RoboDK station: WORKING_EXAMPLE.rdk

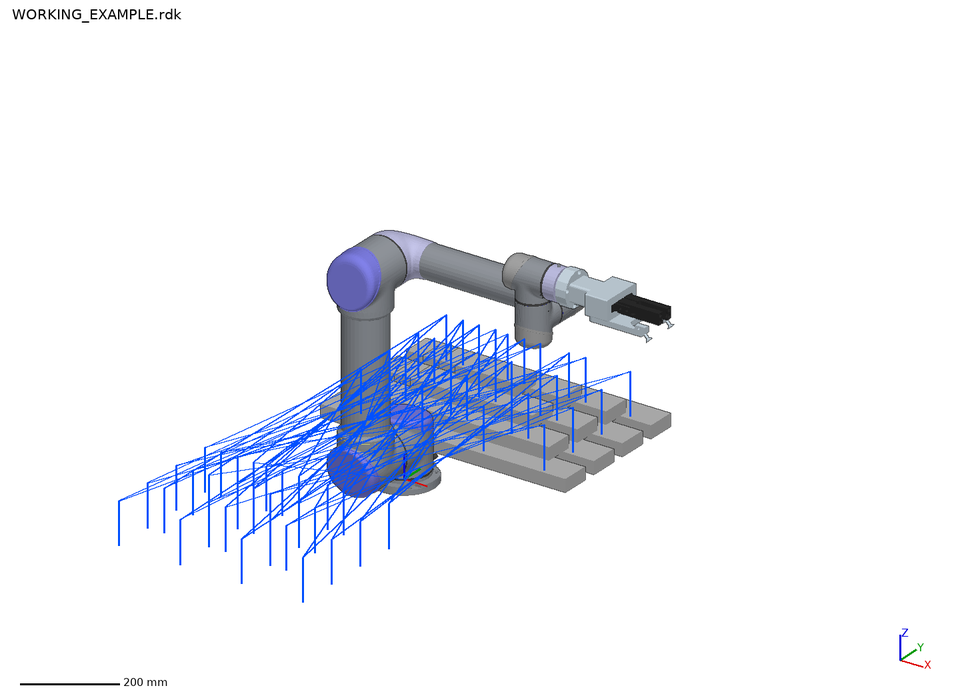
[picture v0: the station drawn from its stored meshes, robots at their saved joint values, targets as dots, program paths as lines]
Station WORKING_EXAMPLE (saved by RoboDK 5.2.1). Poses are relative to the parent item; angles as X-Y-Z fixed-axis rotations.
Station parameters (name, value as stored): Gripper, 0, CollisionFreePlanner, UR5, CollisionFreePlanner-Rob UR5
  - frame UR5 Base at (0, 0, 0) mm
    - robot UR5: 6 axes, payload 5 kg, reach 850 mm, repeatability 0.1 mm, weight 18.4 kg
        modified DH rows (alpha deg, a mm, theta deg, d mm): 0, 0, 0, 89.2; 90, 0, 180, 0; 0, 425, 0, 0; 0, 392.43, 0, 109; -90, 0, 0, 93.65; 90, 0, 180, 82
        joint limits [-360, -180, -180, -360, -360, -360] to [360, 0, 180, 0, 360, 360]; home [0, -90, -90, 0, 90, 0]; saved at [0, -90, -90, 0, 90, 0]
      - tool Gripper, TCP at (0, 0, 240) mm, rotated rx 0 ry 0 rz -90 deg, size 100 x 89.2 x 240.5 mm
    - frame FrameN at (0, 0, 0) mm
      - target csv_data-0 (Cartesian target) at (-26, 357, 183) mm, rotated rx 180 ry 0 rz 180 deg; joints [0, -90, -90, 0, 90, 0] of UR5
      - target csv_data-1 (Cartesian target) at (-26, 357, 83) mm, rotated rx 180 ry 0 rz 180 deg; joints [0, -90, -90, 0, 90, 0] of UR5
      - target csv_data-2 (Cartesian target) at (-26, 357, 183) mm, rotated rx 180 ry 0 rz 180 deg; joints [0, -90, -90, 0, 90, 0] of UR5
      - target csv_data-3 (Cartesian target) at (-301, -567, 93) mm, rotated rx 180 ry 0 rz 180 deg; joints [0, -90, -90, 0, 90, 0] of UR5
      - target csv_data-4 (Cartesian target) at (-301, -567, -7) mm, rotated rx 180 ry 0 rz 180 deg; joints [0, -90, -90, 0, 90, 0] of UR5
      - target csv_data-5 (Cartesian target) at (-301, -567, 93) mm, rotated rx 180 ry 0 rz 180 deg; joints [0, -90, -90, 0, 90, 0] of UR5
      - target csv_data-6 (Cartesian target) at (49, 407, 153) mm, rotated rx 180 ry 0 rz 0 deg; joints [0, -90, -90, 0, 90, 0] of UR5
      - target csv_data-7 (Cartesian target) at (49, 407, 53) mm, rotated rx 180 ry 0 rz 0 deg; joints [0, -90, -90, 0, 90, 0] of UR5
      - target csv_data-8 (Cartesian target) at (49, 407, 153) mm, rotated rx 180 ry 0 rz 0 deg; joints [0, -90, -90, 0, 90, 0] of UR5
      - target csv_data-9 (Cartesian target) at (-151, -567, 93) mm, rotated rx 180 ry 0 rz 180 deg; joints [0, -90, -90, 0, 90, 0] of UR5
      - target csv_data-10 (Cartesian target) at (-151, -567, -7) mm, rotated rx 180 ry 0 rz 180 deg; joints [0, -90, -90, 0, 90, 0] of UR5
      - target csv_data-11 (Cartesian target) at (-151, -567, 93) mm, rotated rx 180 ry 0 rz 180 deg; joints [0, -90, -90, 0, 90, 0] of UR5
      - target csv_data-12 (Cartesian target) at (-101, 407, 153) mm, rotated rx 180 ry 0 rz 180 deg; joints [0, -90, -90, 0, 90, 0] of UR5
      - target csv_data-13 (Cartesian target) at (-101, 407, 53) mm, rotated rx 180 ry 0 rz 180 deg; joints [0, -90, -90, 0, 90, 0] of UR5
      - target csv_data-14 (Cartesian target) at (-101, 407, 153) mm, rotated rx 180 ry 0 rz 180 deg; joints [0, -90, -90, 0, 90, 0] of UR5
      - target csv_data-15 (Cartesian target) at (-1, -567, 93) mm, rotated rx 180 ry 0 rz 180 deg; joints [0, -90, -90, 0, 90, 0] of UR5
      - target csv_data-16 (Cartesian target) at (-1, -567, -7) mm, rotated rx 180 ry 0 rz 180 deg; joints [0, -90, -90, 0, 90, 0] of UR5
      - target csv_data-17 (Cartesian target) at (-1, -567, 93) mm, rotated rx 180 ry 0 rz 180 deg; joints [0, -90, -90, 0, 90, 0] of UR5
      - target csv_data-18 (Cartesian target) at (49, 307, 153) mm, rotated rx 180 ry 0 rz 0 deg; joints [0, -90, -90, 0, 90, 0] of UR5
      - target csv_data-19 (Cartesian target) at (49, 307, 53) mm, rotated rx 180 ry 0 rz 0 deg; joints [0, -90, -90, 0, 90, 0] of UR5
      - target csv_data-20 (Cartesian target) at (49, 307, 153) mm, rotated rx 180 ry 0 rz 0 deg; joints [0, -90, -90, 0, 90, 0] of UR5
      - target csv_data-21 (Cartesian target) at (149, -567, 93) mm, rotated rx 180 ry 0 rz 0 deg; joints [0, -90, -90, 0, 90, 0] of UR5
      - target csv_data-22 (Cartesian target) at (149, -567, -7) mm, rotated rx 180 ry 0 rz 0 deg; joints [0, -90, -90, 0, 90, 0] of UR5
      - target csv_data-23 (Cartesian target) at (149, -567, 93) mm, rotated rx 180 ry 0 rz 0 deg; joints [0, -90, -90, 0, 90, 0] of UR5
      - target csv_data-24 (Cartesian target) at (-101, 307, 153) mm, rotated rx 180 ry 0 rz 180 deg; joints [0, -90, -90, 0, 90, 0] of UR5
      - target csv_data-25 (Cartesian target) at (-101, 307, 53) mm, rotated rx 180 ry 0 rz 180 deg; joints [0, -90, -90, 0, 90, 0] of UR5
      - target csv_data-26 (Cartesian target) at (-101, 307, 153) mm, rotated rx 180 ry 0 rz 180 deg; joints [0, -90, -90, 0, 90, 0] of UR5
      - target csv_data-27 (Cartesian target) at (-301, -467, 93) mm, rotated rx 180 ry 0 rz 180 deg; joints [0, -90, -90, 0, 90, 0] of UR5
      - target csv_data-28 (Cartesian target) at (-301, -467, -7) mm, rotated rx 180 ry 0 rz 180 deg; joints [0, -90, -90, 0, 90, 0] of UR5
      - target csv_data-29 (Cartesian target) at (-301, -467, 93) mm, rotated rx 180 ry 0 rz 180 deg; joints [0, -90, -90, 0, 90, 0] of UR5
      - target csv_data-30 (Cartesian target) at (124, 457, 123) mm, rotated rx 180 ry 0 rz 0 deg; joints [0, -90, -90, 0, 90, 0] of UR5
      - target csv_data-31 (Cartesian target) at (124, 457, 23) mm, rotated rx 180 ry 0 rz 0 deg; joints [0, -90, -90, 0, 90, 0] of UR5
      - target csv_data-32 (Cartesian target) at (124, 457, 123) mm, rotated rx 180 ry 0 rz 0 deg; joints [0, -90, -90, 0, 90, 0] of UR5
      - target csv_data-33 (Cartesian target) at (-151, -467, 93) mm, rotated rx 180 ry 0 rz 180 deg; joints [0, -90, -90, 0, 90, 0] of UR5
      - target csv_data-34 (Cartesian target) at (-151, -467, -7) mm, rotated rx 180 ry 0 rz 180 deg; joints [0, -90, -90, 0, 90, 0] of UR5
      - target csv_data-35 (Cartesian target) at (-151, -467, 93) mm, rotated rx 180 ry 0 rz 180 deg; joints [0, -90, -90, 0, 90, 0] of UR5
      - target csv_data-36 (Cartesian target) at (-26, 457, 123) mm, rotated rx 180 ry 0 rz 180 deg; joints [0, -90, -90, 0, 90, 0] of UR5
      - target csv_data-37 (Cartesian target) at (-26, 457, 23) mm, rotated rx 180 ry 0 rz 180 deg; joints [0, -90, -90, 0, 90, 0] of UR5
      - target csv_data-38 (Cartesian target) at (-26, 457, 123) mm, rotated rx 180 ry 0 rz 180 deg; joints [0, -90, -90, 0, 90, 0] of UR5
      - target csv_data-39 (Cartesian target) at (-1, -467, 93) mm, rotated rx 180 ry 0 rz 180 deg; joints [0, -90, -90, 0, 90, 0] of UR5
      - target csv_data-40 (Cartesian target) at (-1, -467, -7) mm, rotated rx 180 ry 0 rz 180 deg; joints [0, -90, -90, 0, 90, 0] of UR5
      - target csv_data-41 (Cartesian target) at (-1, -467, 93) mm, rotated rx 180 ry 0 rz 180 deg; joints [0, -90, -90, 0, 90, 0] of UR5
      - target csv_data-42 (Cartesian target) at (-176, 457, 123) mm, rotated rx 180 ry 0 rz 180 deg; joints [0, -90, -90, 0, 90, 0] of UR5
      - target csv_data-43 (Cartesian target) at (-176, 457, 23) mm, rotated rx 180 ry 0 rz 180 deg; joints [0, -90, -90, 0, 90, 0] of UR5
      - target csv_data-44 (Cartesian target) at (-176, 457, 123) mm, rotated rx 180 ry 0 rz 180 deg; joints [0, -90, -90, 0, 90, 0] of UR5
      - target csv_data-45 (Cartesian target) at (149, -467, 93) mm, rotated rx 180 ry 0 rz 0 deg; joints [0, -90, -90, 0, 90, 0] of UR5
      - target csv_data-46 (Cartesian target) at (149, -467, -7) mm, rotated rx 180 ry 0 rz 0 deg; joints [0, -90, -90, 0, 90, 0] of UR5
      - target csv_data-47 (Cartesian target) at (149, -467, 93) mm, rotated rx 180 ry 0 rz 0 deg; joints [0, -90, -90, 0, 90, 0] of UR5
      - target csv_data-48 (Cartesian target) at (124, 357, 123) mm, rotated rx 180 ry 0 rz 0 deg; joints [0, -90, -90, 0, 90, 0] of UR5
      - target csv_data-49 (Cartesian target) at (124, 357, 23) mm, rotated rx 180 ry 0 rz 0 deg; joints [0, -90, -90, 0, 90, 0] of UR5
      - target csv_data-50 (Cartesian target) at (124, 357, 123) mm, rotated rx 180 ry 0 rz 0 deg; joints [0, -90, -90, 0, 90, 0] of UR5
      - target csv_data-51 (Cartesian target) at (-301, -367, 93) mm, rotated rx 180 ry 0 rz 180 deg; joints [0, -90, -90, 0, 90, 0] of UR5
      - target csv_data-52 (Cartesian target) at (-301, -367, -7) mm, rotated rx 180 ry 0 rz 180 deg; joints [0, -90, -90, 0, 90, 0] of UR5
      - target csv_data-53 (Cartesian target) at (-301, -367, 93) mm, rotated rx 180 ry 0 rz 180 deg; joints [0, -90, -90, 0, 90, 0] of UR5
      - target csv_data-54 (Cartesian target) at (-26, 357, 123) mm, rotated rx 180 ry 0 rz 180 deg; joints [0, -90, -90, 0, 90, 0] of UR5
      - target csv_data-55 (Cartesian target) at (-26, 357, 23) mm, rotated rx 180 ry 0 rz 180 deg; joints [0, -90, -90, 0, 90, 0] of UR5
      - target csv_data-56 (Cartesian target) at (-26, 357, 123) mm, rotated rx 180 ry 0 rz 180 deg; joints [0, -90, -90, 0, 90, 0] of UR5
      - target csv_data-57 (Cartesian target) at (-151, -367, 93) mm, rotated rx 180 ry 0 rz 180 deg; joints [0, -90, -90, 0, 90, 0] of UR5
      - target csv_data-58 (Cartesian target) at (-151, -367, -7) mm, rotated rx 180 ry 0 rz 180 deg; joints [0, -90, -90, 0, 90, 0] of UR5
      - target csv_data-59 (Cartesian target) at (-151, -367, 93) mm, rotated rx 180 ry 0 rz 180 deg; joints [0, -90, -90, 0, 90, 0] of UR5
      - target csv_data-60 (Cartesian target) at (-176, 357, 123) mm, rotated rx 180 ry 0 rz 180 deg; joints [0, -90, -90, 0, 90, 0] of UR5
      - target csv_data-61 (Cartesian target) at (-176, 357, 23) mm, rotated rx 180 ry 0 rz 180 deg; joints [0, -90, -90, 0, 90, 0] of UR5
      - target csv_data-62 (Cartesian target) at (-176, 357, 123) mm, rotated rx 180 ry 0 rz 180 deg; joints [0, -90, -90, 0, 90, 0] of UR5
      - target csv_data-63 (Cartesian target) at (-1, -367, 93) mm, rotated rx 180 ry 0 rz 180 deg; joints [0, -90, -90, 0, 90, 0] of UR5
      - target csv_data-64 (Cartesian target) at (-1, -367, -7) mm, rotated rx 180 ry 0 rz 180 deg; joints [0, -90, -90, 0, 90, 0] of UR5
      - target csv_data-65 (Cartesian target) at (-1, -367, 93) mm, rotated rx 180 ry 0 rz 180 deg; joints [0, -90, -90, 0, 90, 0] of UR5
      - target csv_data-66 (Cartesian target) at (124, 257, 123) mm, rotated rx 180 ry 0 rz 0 deg; joints [0, -90, -90, 0, 90, 0] of UR5
      - target csv_data-67 (Cartesian target) at (124, 257, 23) mm, rotated rx 180 ry 0 rz 0 deg; joints [0, -90, -90, 0, 90, 0] of UR5
      - target csv_data-68 (Cartesian target) at (124, 257, 123) mm, rotated rx 180 ry 0 rz 0 deg; joints [0, -90, -90, 0, 90, 0] of UR5
      - target csv_data-69 (Cartesian target) at (149, -367, 93) mm, rotated rx 180 ry 0 rz 0 deg; joints [0, -90, -90, 0, 90, 0] of UR5
      - target csv_data-70 (Cartesian target) at (149, -367, -7) mm, rotated rx 180 ry 0 rz 0 deg; joints [0, -90, -90, 0, 90, 0] of UR5
      - target csv_data-71 (Cartesian target) at (149, -367, 93) mm, rotated rx 180 ry 0 rz 0 deg; joints [0, -90, -90, 0, 90, 0] of UR5
      - target csv_data-72 (Cartesian target) at (-26, 257, 123) mm, rotated rx 180 ry 0 rz 180 deg; joints [0, -90, -90, 0, 90, 0] of UR5
      - target csv_data-73 (Cartesian target) at (-26, 257, 23) mm, rotated rx 180 ry 0 rz 180 deg; joints [0, -90, -90, 0, 90, 0] of UR5
      - target csv_data-74 (Cartesian target) at (-26, 257, 123) mm, rotated rx 180 ry 0 rz 180 deg; joints [0, -90, -90, 0, 90, 0] of UR5
      - target csv_data-75 (Cartesian target) at (-301, -267, 93) mm, rotated rx 180 ry 0 rz 180 deg; joints [0, -90, -90, 0, 90, 0] of UR5
      - target csv_data-76 (Cartesian target) at (-301, -267, -7) mm, rotated rx 180 ry 0 rz 180 deg; joints [0, -90, -90, 0, 90, 0] of UR5
      - target csv_data-77 (Cartesian target) at (-301, -267, 93) mm, rotated rx 180 ry 0 rz 180 deg; joints [0, -90, -90, 0, 90, 0] of UR5
      - target csv_data-78 (Cartesian target) at (-176, 257, 123) mm, rotated rx 180 ry 0 rz 180 deg; joints [0, -90, -90, 0, 90, 0] of UR5
      - target csv_data-79 (Cartesian target) at (-176, 257, 23) mm, rotated rx 180 ry 0 rz 180 deg; joints [0, -90, -90, 0, 90, 0] of UR5
      - target csv_data-80 (Cartesian target) at (-176, 257, 123) mm, rotated rx 180 ry 0 rz 180 deg; joints [0, -90, -90, 0, 90, 0] of UR5
      - target csv_data-81 (Cartesian target) at (-151, -267, 93) mm, rotated rx 180 ry 0 rz 180 deg; joints [0, -90, -90, 0, 90, 0] of UR5
      - target csv_data-82 (Cartesian target) at (-151, -267, -7) mm, rotated rx 180 ry 0 rz 180 deg; joints [0, -90, -90, 0, 90, 0] of UR5
      - target csv_data-83 (Cartesian target) at (-151, -267, 93) mm, rotated rx 180 ry 0 rz 180 deg; joints [0, -90, -90, 0, 90, 0] of UR5
      - target csv_data-84 (Cartesian target) at (199, 507, 93) mm, rotated rx 180 ry 0 rz 0 deg; joints [0, -90, -90, 0, 90, 0] of UR5
      - target csv_data-85 (Cartesian target) at (199, 507, -7) mm, rotated rx 180 ry 0 rz 0 deg; joints [0, -90, -90, 0, 90, 0] of UR5
      - target csv_data-86 (Cartesian target) at (199, 507, 93) mm, rotated rx 180 ry 0 rz 0 deg; joints [0, -90, -90, 0, 90, 0] of UR5
      - target csv_data-87 (Cartesian target) at (-1, -267, 93) mm, rotated rx 180 ry 0 rz 180 deg; joints [0, -90, -90, 0, 90, 0] of UR5
      - target csv_data-88 (Cartesian target) at (-1, -267, -7) mm, rotated rx 180 ry 0 rz 180 deg; joints [0, -90, -90, 0, 90, 0] of UR5
      - target csv_data-89 (Cartesian target) at (-1, -267, 93) mm, rotated rx 180 ry 0 rz 180 deg; joints [0, -90, -90, 0, 90, 0] of UR5
      - target csv_data-90 (Cartesian target) at (49, 507, 93) mm, rotated rx 180 ry 0 rz 0 deg; joints [0, -90, -90, 0, 90, 0] of UR5
      - target csv_data-91 (Cartesian target) at (49, 507, -7) mm, rotated rx 180 ry 0 rz 0 deg; joints [0, -90, -90, 0, 90, 0] of UR5
      - target csv_data-92 (Cartesian target) at (49, 507, 93) mm, rotated rx 180 ry 0 rz 0 deg; joints [0, -90, -90, 0, 90, 0] of UR5
      - target csv_data-93 (Cartesian target) at (149, -267, 93) mm, rotated rx 180 ry 0 rz 0 deg; joints [0, -90, -90, 0, 90, 0] of UR5
      - target csv_data-94 (Cartesian target) at (149, -267, -7) mm, rotated rx 180 ry 0 rz 0 deg; joints [0, -90, -90, 0, 90, 0] of UR5
      - target csv_data-95 (Cartesian target) at (149, -267, 93) mm, rotated rx 180 ry 0 rz 0 deg; joints [0, -90, -90, 0, 90, 0] of UR5
      - target csv_data-96 (Cartesian target) at (-101, 507, 93) mm, rotated rx 180 ry 0 rz 180 deg; joints [0, -90, -90, 0, 90, 0] of UR5
      - target csv_data-97 (Cartesian target) at (-101, 507, -7) mm, rotated rx 180 ry 0 rz 180 deg; joints [0, -90, -90, 0, 90, 0] of UR5
      - target csv_data-98 (Cartesian target) at (-101, 507, 93) mm, rotated rx 180 ry 0 rz 180 deg; joints [0, -90, -90, 0, 90, 0] of UR5
      - target csv_data-99 (Cartesian target) at (-226, -517, 123) mm, rotated rx 180 ry 0 rz 180 deg; joints [0, -90, -90, 0, 90, 0] of UR5
      - target csv_data-100 (Cartesian target) at (-226, -517, 23) mm, rotated rx 180 ry 0 rz 180 deg; joints [0, -90, -90, 0, 90, 0] of UR5
      - target csv_data-101 (Cartesian target) at (-226, -517, 123) mm, rotated rx 180 ry 0 rz 180 deg; joints [0, -90, -90, 0, 90, 0] of UR5
      - target csv_data-102 (Cartesian target) at (-251, 507, 93) mm, rotated rx 180 ry 0 rz 180 deg; joints [0, -90, -90, 0, 90, 0] of UR5
      - target csv_data-103 (Cartesian target) at (-251, 507, -7) mm, rotated rx 180 ry 0 rz 180 deg; joints [0, -90, -90, 0, 90, 0] of UR5
      - target csv_data-104 (Cartesian target) at (-251, 507, 93) mm, rotated rx 180 ry 0 rz 180 deg; joints [0, -90, -90, 0, 90, 0] of UR5
      - target csv_data-105 (Cartesian target) at (-76, -517, 123) mm, rotated rx 180 ry 0 rz 180 deg; joints [0, -90, -90, 0, 90, 0] of UR5
      - target csv_data-106 (Cartesian target) at (-76, -517, 23) mm, rotated rx 180 ry 0 rz 180 deg; joints [0, -90, -90, 0, 90, 0] of UR5
      - target csv_data-107 (Cartesian target) at (-76, -517, 123) mm, rotated rx 180 ry 0 rz 180 deg; joints [0, -90, -90, 0, 90, 0] of UR5
      - target csv_data-108 (Cartesian target) at (199, 407, 93) mm, rotated rx 180 ry 0 rz 0 deg; joints [0, -90, -90, 0, 90, 0] of UR5
      - target csv_data-109 (Cartesian target) at (199, 407, -7) mm, rotated rx 180 ry 0 rz 0 deg; joints [0, -90, -90, 0, 90, 0] of UR5
      - target csv_data-110 (Cartesian target) at (199, 407, 93) mm, rotated rx 180 ry 0 rz 0 deg; joints [0, -90, -90, 0, 90, 0] of UR5
      - target csv_data-111 (Cartesian target) at (74, -517, 123) mm, rotated rx 180 ry 0 rz 0 deg; joints [0, -90, -90, 0, 90, 0] of UR5
      - target csv_data-112 (Cartesian target) at (74, -517, 23) mm, rotated rx 180 ry 0 rz 0 deg; joints [0, -90, -90, 0, 90, 0] of UR5
      - target csv_data-113 (Cartesian target) at (74, -517, 123) mm, rotated rx 180 ry 0 rz 0 deg; joints [0, -90, -90, 0, 90, 0] of UR5
      - target csv_data-114 (Cartesian target) at (49, 407, 93) mm, rotated rx 180 ry 0 rz 0 deg; joints [0, -90, -90, 0, 90, 0] of UR5
      - target csv_data-115 (Cartesian target) at (49, 407, -7) mm, rotated rx 180 ry 0 rz 0 deg; joints [0, -90, -90, 0, 90, 0] of UR5
      - target csv_data-116 (Cartesian target) at (49, 407, 93) mm, rotated rx 180 ry 0 rz 0 deg; joints [0, -90, -90, 0, 90, 0] of UR5
      - target csv_data-117 (Cartesian target) at (-226, -417, 123) mm, rotated rx 180 ry 0 rz 180 deg; joints [0, -90, -90, 0, 90, 0] of UR5
      - target csv_data-118 (Cartesian target) at (-226, -417, 23) mm, rotated rx 180 ry 0 rz 180 deg; joints [0, -90, -90, 0, 90, 0] of UR5
      - target csv_data-119 (Cartesian target) at (-226, -417, 123) mm, rotated rx 180 ry 0 rz 180 deg; joints [0, -90, -90, 0, 90, 0] of UR5
      - target csv_data-120 (Cartesian target) at (-101, 407, 93) mm, rotated rx 180 ry 0 rz 180 deg; joints [0, -90, -90, 0, 90, 0] of UR5
      - target csv_data-121 (Cartesian target) at (-101, 407, -7) mm, rotated rx 180 ry 0 rz 180 deg; joints [0, -90, -90, 0, 90, 0] of UR5
      - target csv_data-122 (Cartesian target) at (-101, 407, 93) mm, rotated rx 180 ry 0 rz 180 deg; joints [0, -90, -90, 0, 90, 0] of UR5
      - target csv_data-123 (Cartesian target) at (-76, -417, 123) mm, rotated rx 180 ry 0 rz 180 deg; joints [0, -90, -90, 0, 90, 0] of UR5
      - target csv_data-124 (Cartesian target) at (-76, -417, 23) mm, rotated rx 180 ry 0 rz 180 deg; joints [0, -90, -90, 0, 90, 0] of UR5
      - target csv_data-125 (Cartesian target) at (-76, -417, 123) mm, rotated rx 180 ry 0 rz 180 deg; joints [0, -90, -90, 0, 90, 0] of UR5
      - target csv_data-126 (Cartesian target) at (-251, 407, 93) mm, rotated rx 180 ry 0 rz 180 deg; joints [0, -90, -90, 0, 90, 0] of UR5
      - target csv_data-127 (Cartesian target) at (-251, 407, -7) mm, rotated rx 180 ry 0 rz 180 deg; joints [0, -90, -90, 0, 90, 0] of UR5
      - target csv_data-128 (Cartesian target) at (-251, 407, 93) mm, rotated rx 180 ry 0 rz 180 deg; joints [0, -90, -90, 0, 90, 0] of UR5
      - target csv_data-129 (Cartesian target) at (74, -417, 123) mm, rotated rx 180 ry 0 rz 0 deg; joints [0, -90, -90, 0, 90, 0] of UR5
      - target csv_data-130 (Cartesian target) at (74, -417, 23) mm, rotated rx 180 ry 0 rz 0 deg; joints [0, -90, -90, 0, 90, 0] of UR5
      - target csv_data-131 (Cartesian target) at (74, -417, 123) mm, rotated rx 180 ry 0 rz 0 deg; joints [0, -90, -90, 0, 90, 0] of UR5
      - target csv_data-132 (Cartesian target) at (199, 307, 93) mm, rotated rx 180 ry 0 rz 0 deg; joints [0, -90, -90, 0, 90, 0] of UR5
      - target csv_data-133 (Cartesian target) at (199, 307, -7) mm, rotated rx 180 ry 0 rz 0 deg; joints [0, -90, -90, 0, 90, 0] of UR5
      - target csv_data-134 (Cartesian target) at (199, 307, 93) mm, rotated rx 180 ry 0 rz 0 deg; joints [0, -90, -90, 0, 90, 0] of UR5
      - target csv_data-135 (Cartesian target) at (-226, -317, 123) mm, rotated rx 180 ry 0 rz 180 deg; joints [0, -90, -90, 0, 90, 0] of UR5
      - target csv_data-136 (Cartesian target) at (-226, -317, 23) mm, rotated rx 180 ry 0 rz 180 deg; joints [0, -90, -90, 0, 90, 0] of UR5
      - target csv_data-137 (Cartesian target) at (-226, -317, 123) mm, rotated rx 180 ry 0 rz 180 deg; joints [0, -90, -90, 0, 90, 0] of UR5
      - target csv_data-138 (Cartesian target) at (49, 307, 93) mm, rotated rx 180 ry 0 rz 0 deg; joints [0, -90, -90, 0, 90, 0] of UR5
      - target csv_data-139 (Cartesian target) at (49, 307, -7) mm, rotated rx 180 ry 0 rz 0 deg; joints [0, -90, -90, 0, 90, 0] of UR5
      - target csv_data-140 (Cartesian target) at (49, 307, 93) mm, rotated rx 180 ry 0 rz 0 deg; joints [0, -90, -90, 0, 90, 0] of UR5
      - target csv_data-141 (Cartesian target) at (-76, -317, 123) mm, rotated rx 180 ry 0 rz 180 deg; joints [0, -90, -90, 0, 90, 0] of UR5
      - target csv_data-142 (Cartesian target) at (-76, -317, 23) mm, rotated rx 180 ry 0 rz 180 deg; joints [0, -90, -90, 0, 90, 0] of UR5
      - target csv_data-143 (Cartesian target) at (-76, -317, 123) mm, rotated rx 180 ry 0 rz 180 deg; joints [0, -90, -90, 0, 90, 0] of UR5
      - target csv_data-144 (Cartesian target) at (-101, 307, 93) mm, rotated rx 180 ry 0 rz 180 deg; joints [0, -90, -90, 0, 90, 0] of UR5
      - target csv_data-145 (Cartesian target) at (-101, 307, -7) mm, rotated rx 180 ry 0 rz 180 deg; joints [0, -90, -90, 0, 90, 0] of UR5
      - target csv_data-146 (Cartesian target) at (-101, 307, 93) mm, rotated rx 180 ry 0 rz 180 deg; joints [0, -90, -90, 0, 90, 0] of UR5
      - target csv_data-147 (Cartesian target) at (74, -317, 123) mm, rotated rx 180 ry 0 rz 0 deg; joints [0, -90, -90, 0, 90, 0] of UR5
      - target csv_data-148 (Cartesian target) at (74, -317, 23) mm, rotated rx 180 ry 0 rz 0 deg; joints [0, -90, -90, 0, 90, 0] of UR5
      - target csv_data-149 (Cartesian target) at (74, -317, 123) mm, rotated rx 180 ry 0 rz 0 deg; joints [0, -90, -90, 0, 90, 0] of UR5
      - target csv_data-150 (Cartesian target) at (-251, 307, 93) mm, rotated rx 180 ry 0 rz 180 deg; joints [0, -90, -90, 0, 90, 0] of UR5
      - target csv_data-151 (Cartesian target) at (-251, 307, -7) mm, rotated rx 180 ry 0 rz 180 deg; joints [0, -90, -90, 0, 90, 0] of UR5
      - target csv_data-152 (Cartesian target) at (-251, 307, 93) mm, rotated rx 180 ry 0 rz 180 deg; joints [0, -90, -90, 0, 90, 0] of UR5
      - target csv_data-153 (Cartesian target) at (-151, -467, 153) mm, rotated rx 180 ry 0 rz 180 deg; joints [0, -90, -90, 0, 90, 0] of UR5
      - target csv_data-154 (Cartesian target) at (-151, -467, 53) mm, rotated rx 180 ry 0 rz 180 deg; joints [0, -90, -90, 0, 90, 0] of UR5
      - target csv_data-155 (Cartesian target) at (-151, -467, 153) mm, rotated rx 180 ry 0 rz 180 deg; joints [0, -90, -90, 0, 90, 0] of UR5
      - target csv_data-156 (Cartesian target) at (199, 207, 93) mm, rotated rx 180 ry 0 rz 0 deg; joints [0, -90, -90, 0, 90, 0] of UR5
      - target csv_data-157 (Cartesian target) at (199, 207, -7) mm, rotated rx 180 ry 0 rz 0 deg; joints [0, -90, -90, 0, 90, 0] of UR5
      - target csv_data-158 (Cartesian target) at (199, 207, 93) mm, rotated rx 180 ry 0 rz 0 deg; joints [0, -90, -90, 0, 90, 0] of UR5
      - target csv_data-159 (Cartesian target) at (-1, -467, 153) mm, rotated rx 180 ry 0 rz 180 deg; joints [0, -90, -90, 0, 90, 0] of UR5
      - target csv_data-160 (Cartesian target) at (-1, -467, 53) mm, rotated rx 180 ry 0 rz 180 deg; joints [0, -90, -90, 0, 90, 0] of UR5
      - target csv_data-161 (Cartesian target) at (-1, -467, 153) mm, rotated rx 180 ry 0 rz 180 deg; joints [0, -90, -90, 0, 90, 0] of UR5
      - target csv_data-162 (Cartesian target) at (49, 207, 93) mm, rotated rx 180 ry 0 rz 0 deg; joints [0, -90, -90, 0, 90, 0] of UR5
      - target csv_data-163 (Cartesian target) at (49, 207, -7) mm, rotated rx 180 ry 0 rz 0 deg; joints [0, -90, -90, 0, 90, 0] of UR5
      - target csv_data-164 (Cartesian target) at (49, 207, 93) mm, rotated rx 180 ry 0 rz 0 deg; joints [0, -90, -90, 0, 90, 0] of UR5
      - target csv_data-165 (Cartesian target) at (-151, -367, 153) mm, rotated rx 180 ry 0 rz 180 deg; joints [0, -90, -90, 0, 90, 0] of UR5
      - target csv_data-166 (Cartesian target) at (-151, -367, 53) mm, rotated rx 180 ry 0 rz 180 deg; joints [0, -90, -90, 0, 90, 0] of UR5
      - target csv_data-167 (Cartesian target) at (-151, -367, 153) mm, rotated rx 180 ry 0 rz 180 deg; joints [0, -90, -90, 0, 90, 0] of UR5
      - target csv_data-168 (Cartesian target) at (-101, 207, 93) mm, rotated rx 180 ry 0 rz 180 deg; joints [0, -90, -90, 0, 90, 0] of UR5
      - target csv_data-169 (Cartesian target) at (-101, 207, -7) mm, rotated rx 180 ry 0 rz 180 deg; joints [0, -90, -90, 0, 90, 0] of UR5
      - target csv_data-170 (Cartesian target) at (-101, 207, 93) mm, rotated rx 180 ry 0 rz 180 deg; joints [0, -90, -90, 0, 90, 0] of UR5
      - target csv_data-171 (Cartesian target) at (-1, -367, 153) mm, rotated rx 180 ry 0 rz 180 deg; joints [0, -90, -90, 0, 90, 0] of UR5
      - target csv_data-172 (Cartesian target) at (-1, -367, 53) mm, rotated rx 180 ry 0 rz 180 deg; joints [0, -90, -90, 0, 90, 0] of UR5
      - target csv_data-173 (Cartesian target) at (-1, -367, 153) mm, rotated rx 180 ry 0 rz 180 deg; joints [0, -90, -90, 0, 90, 0] of UR5
      - target csv_data-174 (Cartesian target) at (-251, 207, 93) mm, rotated rx 180 ry 0 rz 180 deg; joints [0, -90, -90, 0, 90, 0] of UR5
      - target csv_data-175 (Cartesian target) at (-251, 207, -7) mm, rotated rx 180 ry 0 rz 180 deg; joints [0, -90, -90, 0, 90, 0] of UR5
      - target csv_data-176 (Cartesian target) at (-251, 207, 93) mm, rotated rx 180 ry 0 rz 180 deg; joints [0, -90, -90, 0, 90, 0] of UR5
      - target csv_data-177 (Cartesian target) at (-76, -417, 183) mm, rotated rx 180 ry 0 rz 180 deg; joints [0, -90, -90, 0, 90, 0] of UR5
      - target csv_data-178 (Cartesian target) at (-76, -417, 83) mm, rotated rx 180 ry 0 rz 180 deg; joints [0, -90, -90, 0, 90, 0] of UR5
      - target csv_data-179 (Cartesian target) at (-76, -417, 183) mm, rotated rx 180 ry 0 rz 180 deg; joints [0, -90, -90, 0, 90, 0] of UR5
    - object Table at (-250, 600, 0) mm, rotated rx 0 ry 0 rz -180 deg, size 600 x 1350 x 100 mm, geometry from RhinoPart.ply
    - object Closed Brep_0 at (0, 0, 0) mm, size 150 x 70 x 30 mm
    - object Closed Brep_1 at (0, 0, 0) mm, size 150 x 70 x 30 mm
    - object Closed Brep_2 at (0, 0, 0) mm, size 150 x 70 x 30 mm
    - object Closed Brep_3 at (0, 0, 0) mm, size 150 x 70 x 30 mm
    - object Closed Brep_4 at (0, 0, 0) mm, size 150 x 70 x 30 mm
    - object Closed Brep_5 at (0, 0, 0) mm, size 150 x 70 x 30 mm
    - object Closed Brep_6 at (0, 0, 0) mm, size 150 x 70 x 30 mm
    - object Closed Brep_7 at (0, 0, 0) mm, size 150 x 70 x 30 mm
    - object Closed Brep_8 at (0, 0, 0) mm, size 150 x 70 x 30 mm
    - object Closed Brep_9 at (0, 0, 0) mm, size 150 x 70 x 30 mm
    - object Closed Brep_10 at (0, 0, 0) mm, size 150 x 70 x 30 mm
    - object Closed Brep_11 at (0, 0, 0) mm, size 150 x 70 x 30 mm
    - object Closed Brep_12 at (0, 0, 0) mm, size 150 x 70 x 30 mm
    - object Closed Brep_13 at (0, 0, 0) mm, size 150 x 70 x 30 mm
    - object Closed Brep_14 at (0, 0, 0) mm, size 150 x 70 x 30 mm
    - object Closed Brep_15 at (0, 0, 0) mm, size 150 x 70 x 30 mm
    - object Closed Brep_16 at (0, 0, 0) mm, size 150 x 70 x 30 mm
    - object Closed Brep_17 at (0, 0, 0) mm, size 150 x 70 x 30 mm
    - object Closed Brep_18 at (0, 0, 0) mm, size 150 x 70 x 30 mm
    - object Closed Brep_19 at (0, 0, 0) mm, size 150 x 70 x 30 mm
    - object Closed Brep_20 at (0, 0, 0) mm, size 150 x 70 x 30 mm
    - object Closed Brep_21 at (0, 0, 0) mm, size 150 x 70 x 30 mm
    - object Closed Brep_22 at (0, 0, 0) mm, size 150 x 70 x 30 mm
    - object Closed Brep_23 at (0, 0, 0) mm, size 150 x 70 x 30 mm
    - object Closed Brep_24 at (0, 0, 0) mm, size 150 x 70 x 30 mm
    - object Closed Brep_25 at (0, 0, 0) mm, size 150 x 70 x 30 mm
    - object Closed Brep_26 at (0, 0, 0) mm, size 150 x 70 x 30 mm
    - object Closed Brep_27 at (0, 0, 0) mm, size 150 x 70 x 30 mm
    - object Closed Brep_28 at (0, 0, 0) mm, size 150 x 70 x 30 mm
    - object Closed Brep_29 at (0, 0, 0) mm, size 150 x 70 x 30 mm
  - Python program Generate_csv_program (listed below)
  - Python program Import_Rhino_geometry (listed below)
  - program Main_Program (365 instructions, listed below)
  - program Attach (3 instructions, listed below)
  - program Detach (3 instructions, listed below)
  - program Return_Bricks (1 instructions, listed below)
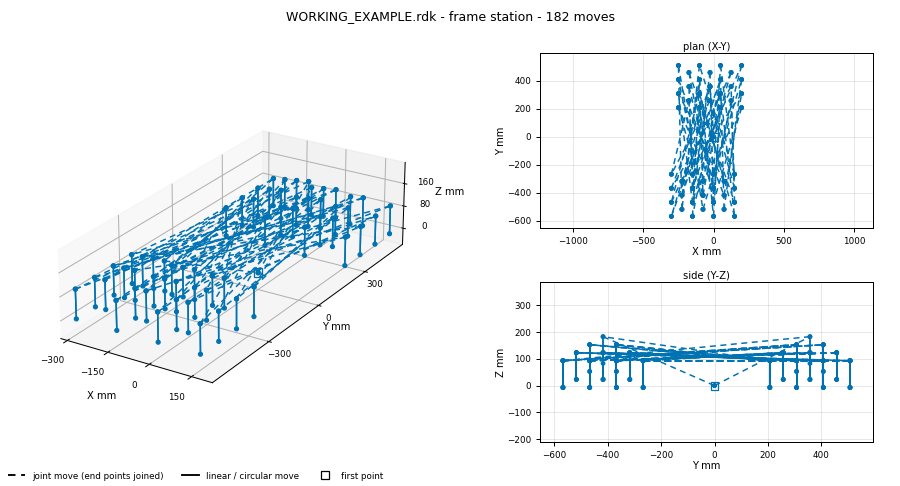
[picture p0: tool path of WORKING_EXAMPLE.rdk in frame station, 182 of 182 moves have a stored position in this frame; points joined in program order, loops and branches not executed]

--- Python program Generate_csv_program ---
# This macro can load CSV files in RoboDK. It also allows the user
# Supported types of files are:
#  1-Tool data : Tool.csv
#  2-Work object data: Work.csv
#  3-Target data: P_Var.csv
# This macro can also filter a given targets file

# Type help("robolink") or help("robodk") for more information
# Press F5 to run the script
# Visit: http://www.robodk.com/doc/PythonAPI/
# For RoboDK API documentation

# This script has been further developed by Job de Vogel
# It is based on the example ImportCSV_XYZWPR.py script

from robolink import *    # API to communicate with RoboDK
from robodk import *      # basic matrix operations

# Start communication with RoboDK
RDK = Robolink()

# Ask the user to select the robot (ignores the popup if only
ROBOT = RDK.ItemUserPick('Select a robot', ITEM_TYPE_ROBOT)

# Check if the user selected a robot
if not ROBOT.Valid():
    quit()

# Automatically retrieve active reference and tool
FRAME = ROBOT.getLink(ITEM_TYPE_FRAME)
TOOL = ROBOT.getLink(ITEM_TYPE_TOOL)

#FRAME = RDK.ItemUserPick('Select a reference frame', ITEM_TYPE_FRAME)
#TOOL = RDK.ItemUserPick('Select a tool', ITEM_TYPE_TOOL)

if not FRAME.Valid() or not TOOL.Valid():
    raise Exception("Select appropriate FRAME and TOOL references")

# Function to convert XYZWPR to a pose
# Important! Specify the order of rotation
def xyzwpr_to_pose(xyzwpr):
    x,y,z,rx,ry,rz = xyzwpr
    return transl(x,y,z)*rotz(rz*pi/180)*roty(ry*pi/180)*rotx(rx*pi/180)
    #return transl(x,y,z)*rotx(rx*pi/180)*roty(ry*pi/180)*rotz(rz*pi/180)
    #return KUKA_2_Pose(xyzwpr)

# Load P_Var.CSV data as a list of poses, including links to reference and tool frames
def load_targets(strfile):
    csvdata = LoadList(strfile, ',', codec)

    idxs = [] # row index of the csv data
    poses = [] # pose of the csv data, based on x,y,z,rx,ry,rz
    movetypes = [] # type of movement: linear (l) or joint (j)
    speeds = [] # joint speed of the robot
    subprogram_names = []

    """ EXTRACT EXTRA DATA
    HERE YOU INITIALIZE EXTRA VARIABLES THAT THE CSV DATA CONTAINS
    """

    # Iterate over the rows with instructions in the csv
    for i in range(0, len(csvdata)):
        # Extract the index of the instruction
        idxs.append(i)

        # Extract the pose data from the csv
        try:
            x,y,z,rx,ry,rz = csvdata[i][0:6]
            poses.append(xyzwpr_to_pose([x,y,z,rx,ry,rz]))
        except:
            print("No pose available to extract")
            return

        # Extract the speed data from the csv
        try:
            speed = csvdata[i][6]
            speeds.append(speed)
        except:
            speeds.append("")

        # Extract the movetypes from the csv
        try:
            movetype = csvdata[i][7]
            movetypes.append(movetype)
        except IndexError:
            movetypes.append("")

        # Extract the subprograms from the csv
        try:
            subprogram = csvdata[i][8]
            subprogram_names.append(subprogram)
        except:
            subprogram_names.append("")

        """ADD DATA
        HERE YOU EXTRACT OTHER DATA FROM THE CSV
        MAKE SURE YOU RETURN THE DATA AT THE END OF THIS DEFINITION

        ALWAYS ADD A TRY-EXCEPT STATEMENT IN CASE NO DATA IS
        AVAILABLE IN THE CSV
        """

    return idxs, poses, movetypes, speeds, subprogram_names

# Load the data from the CSV and add the instruction to the main program
def load_program_csv(strfile, program_name):
    # Get the data from .csv
    idxs, poses, movetypes, speeds, subprogram_names = load_targets(strfile)

    # Set the name for the csv
    csv_name = getFileName(strfile)
    csv_name = csv_name.replace('-','_').replace(' ','_')

    # Create a RDK program item
    program = RDK.Item(program_name, ITEM_TYPE_PROGRAM)

    # If the program already exists, delete it
    if program.Valid():
        program.Delete()

    # Add the main program to the robot
    program = RDK.AddProgram(program_name, ROBOT)

    # Set the frame and the tool to the main program
    program.setFrame(FRAME)
    program.setTool(TOOL)

    # Move the robot home
    ROBOT.MoveJ(ROBOT.JointsHome())
    program.MoveJ(ROBOT.JointsHome())

    # For each point from the csv, add the following instuction to the main program
    for idx, pose, movetype, speed, subprogram_name in zip(idxs, poses, movetypes, speeds, subprogram_names):

        #status = program.Update(1)
        #print(status)

        # Set the name of the point
        name = '%s-%i' % (csv_name, idx)

        # Create a target for the name
        target = RDK.Item(name, ITEM_TYPE_TARGET)

        # If the target already exists, delete it
        if target.Valid():
            target.Delete()

        # Add the target to the main program
        target = RDK.AddTarget(name, FRAME, ROBOT)
        target.setPose(pose)

        """ ADD INSTRUCTIONS
        FROM HERE ON, THE ROBOT WILL ADD THE INSTRUCTION FROM THE CSV TO THE PROGRAM
        CURRENTLY, THE INSTRUCTIONS ARE ADDED ACCORDING THE ORDER OF THE CSV COLUMNS
        """

        # Add the movement to the program
        # Overwrite to joint to avoid singularities:
        if movetype == "linear":
            try:
                program.MoveL(target)
            except:
                print('Warning: {} can not be reached. It will not be added to the program'.format(name))
        else:
            try:
                program.MoveJ(target)
            except:
                print('Warning: {} can not be reached. It will not be added to the program'.format(name))

        # Set a speed for the robot
        if speed:
            program.setSpeed(speed, speed)

        # Check if this csv row has a subprogram to run
        if subprogram_name:
            subprogram = RDK.Item(subprogram_name, ITEM_TYPE_PROGRAM)

            # If the subprogram does not yet exist, add it to the Robot tree
            if not subprogram.Valid():
                subprogram = RDK.AddProgram(subprogram_name, ROBOT)
                print("{} added to Robot".format(subprogram_name))

            program.RunInstruction(subprogram_name)

        """TO ADD INSTRUCTIONS:
        FROM HERE ON, YOU CAN ADD YOUR OWN INSTRUCTIONS TO THE ROBOT
        MAKE SURE YOU ADD THEM IN THE CORRECT ORDER

        TAKE A LOOK AT https://robodk.com/doc/en/PythonAPI/robolink.html TO SEE WHAT IS POSSIBLE
        """

    # Move the robot home
    program.MoveJ(ROBOT.JointsHome())
    print("{} has been updated!".format(program_name))

# Run the robot simulation
# The run_simulation function does the same as load_program_csv but it doesn't load the program
# to RoboDK. If you only want the Robot to do something, use ROBOT.function() instead of program.function()
# If the program already exists in the tree, it will directly use those instructions,
# to make use of collision detection
def run_simulation(strfile, program_name):
    # Load the data from the csv file
    idxs, poses, movetypes, speeds, subprogram_names = load_targets(strfile)

    # Set the frame and tool of the robot
    ROBOT.setFrame(FRAME)
    ROBOT.setTool(TOOL)

    # Return to home
    ROBOT.MoveJ(ROBOT.JointsHome())

    # Check if program is already added to the robot tree
    # If that is the case, run the instructions directly from the tree
    # Else, robot may execute script without proper collision avoidance
    program = RDK.Item(program_name, ITEM_TYPE_PROGRAM)
    if program.Valid():
        program.RunCode()
        return

    for idx, pose, movetype, speed, subprogram_name in zip(idxs, poses, movetypes, speeds, subprogram_names):
        # Move the robot according to movetype, if no movetype available, do a joint move
        # Overwrite to joint to avoid singularities:
        if movetype == "linear":
            try:
                ROBOT.MoveL(pose)
            except TargetReachError:
                RDK.ShowMessage('Target %i can not be reached' % idx, False)
        else:
            try:
                ROBOT.MoveJ(pose)
            except TargetReachError:
                RDK.ShowMessage('Target %i can not be reached' % idx, False)

        """
        IF YOU ADD INSTRUCTIONS TO THE LOAD_PROGRAM_CSV FUNCTION,
        YOU WILL ALSO NEED TO ADD THEM TO THE RUN_SIMULATION FUNCTION.
        """

        # If there is a speed available, set the linear and joint speed
        if speed:
            print("Set speed to {} m/s".format(speed))
            ROBOT.setSpeed(speed, speed)

        # If a subprogram should be run, run the subprogram
        if subprogram_name:
            subprogram = RDK.Item(subprogram_name, ITEM_TYPE_PROGRAM)

            if subprogram.Valid():
                print("Robot is running {}".format(subprogram_name))
                subprogram.RunCode()
            else:
                print("{} is not valid, the subprogram will be skipped".format(subprogram_name))

    # Return to home
    ROBOT.MoveJ(ROBOT.JointsHome())

######################################### -- MAIN -- ################################################
# Force just moving the robot after double clicking:
#load_targets_move(CSV_FILE)
#quit()

# Specify file codec
codec = 'utf-8' #'ISO-8859-1'

# SPECIFY YOU CSV FILE HERE:
CSV_FILE = r"" # Make sure you add r in front of your string to get a raw string as filepath
SELECT_CSV = mbox('Please select your csv file, you can also specify your csv directory in the generate_csv_program script (line 266)', 'Select')

if SELECT_CSV and not CSV_FILE:
    # No CSV has been specified in line 266, select manually
    CSV_FILE = getOpenFile(RDK.getParam('PATH_OPENSTATION'))
elif not SELECT_CSV and not CSV_FILE:
    # User wants to cancel
    quit()

# PROGRAM/SIMULATION SETTINGS:
MAKE_GUI_PROGRAM = False
SIMULATION_SPEED = 1
PROGRAM_NAME = "Main_Program"

ROBOT.setFrame(FRAME)
ROBOT.setTool(TOOL)

RDK.setSimulationSpeed(SIMULATION_SPEED)

if RDK.RunMode() == RUNMODE_SIMULATE:
    MAKE_GUI_PROGRAM = True
    if CSV_FILE:
        MAKE_GUI_PROGRAM = mbox('Do you want to create a new program? If not, the robot will execute a simulation. If the program does not exist in the RoboDK, collisions may occur!', 'Yes', 'No')
else:
    # If we run in program generation mode just move the robot
    MAKE_GUI_PROGRAM = False

if MAKE_GUI_PROGRAM:
    RDK.Render(False) # Faster if we turn render off
    load_program_csv(CSV_FILE, PROGRAM_NAME) # HERE THE CSV DATA IS LOADED!!!
else:
    run_simulation(CSV_FILE, PROGRAM_NAME) # HERE WE START RUNNING THE PROJECT!!!

--- Python program Import_Rhino_geometry ---
# Type help("robolink") or help("robodk") for more information
# Press F5 to run the script
# Documentation: https://robodk.com/doc/en/RoboDK-API.html
# Reference:     https://robodk.com/doc/en/PythonAPI/index.html

# This script has been developed by Job de Vogel
from robolink import *    # RoboDK API
from robodk import *      # Robot toolbox

RDK = Robolink()

# Ask the user to select the robot (ignores the popup if only
ROBOT = RDK.ItemUserPick('Select a robot', ITEM_TYPE_ROBOT)

# Check if the user selected a robot
if not ROBOT.Valid():
    quit()

# Read the csv with geometry
# First column in csv indicates type (v: vertex, o: order, n: name)
def load_csv_data(strfile):
    csv_file = LoadList(strfile, ',', codec)

    # Store the vertex data, vertex order and name in dict
    vertex_data = {}
    vertex_order = {}
    names = {}

    # For every csv line, check the data type and store value accordingly
    i = 0
    for line in csv_file:
        # Check if geom key in dict contains list, if not create it
        try:
            data = vertex_data[i]
            data = vertex_order[i]
        except KeyError:
            vertex_data[i] = []
            vertex_order[i] = []

        datatype = line[0]
        if datatype == 'v':
            vertex_data[i].append(line[1:])
        elif datatype == 'o':
            vertex_order[i].append(line[1:])
        elif datatype == 'n':
            names[i] = line[1]
            i +=1

    return vertex_data, vertex_order, names

# Create a list that contains all the vertices according to the vertexorder of the shape
def structure_vertexData(vertex_data: list, vertex_order: list):
    data = []
    for order in vertex_order:
        for vertex in order:
            data.append(vertex_data[int(vertex)])

    return data

# Create an RDK item that contains the shape
# The function will copy the shape to clipboard, it can be later pasted to frame using frame.Paste()
def create_shape(name, vertices):
    obj = RDK.Item(name, ITEM_TYPE_OBJECT)

    # If obj already exist, delete previous version
    if obj.Valid():
        obj.Delete()

    # Create a new shape for the obj
    obj = obj.AddShape(vertices)
    obj.setName(name)

    # Copy to paste after return
    obj.Copy()
    obj.Delete()
    return

######################################### -- MAIN -- ################################################
# Specify file codec
codec = 'utf-8' #'ISO-8859-1'

# SPECIFY YOU CSV FILE HERE:
objects_csv_file = r"" # Make sure you add r in front of your string to get a raw string for your filepath
SELECT_CSV = mbox('Please select your csv file that contains your geometry data and frame data. (You can also specify a path in the script in line 83)', 'Select')

if SELECT_CSV and not objects_csv_file:
    # No CSV has been specified in line 83, select manually
    objects_csv_file = getOpenFile(RDK.getParam('PATH_OPENSTATION'))

    if not objects_csv_file:
        quit()
elif not SELECT_CSV and not objects_csv_file:
    # User does not wants to cancel
    quit()

# HERE YOU CAN DEFINE WHERE THE OBJECTS SHOULD BE PASTED:
frame_name = 'UR5 Base' # Name of the frame where your geometry should be added
ROBOT_frame = RDK.Item(frame_name, ITEM_TYPE_FRAME)

if ROBOT_frame.Valid():
    mbox('Your geometry will be added to {}. You can change the frame in script line 97.'.format(frame_name), 'Okay')
else:
    ROBOT.getLink(ITEM_TYPE_FRAME)
    mbox('Your selected frame does not exist in the tree. Frame will be changed to standard Robot frame. Please change in script line 97.', 'Okay')

# Load the geometry csv
geometries = load_csv_data(objects_csv_file)

vertex_data = geometries[0].values()
vertex_order = geometries[1].values()
geom_names = geometries[2].values()

for i, (vertices, indices, geom_name) in enumerate(zip(vertex_data, vertex_order, geom_names)):
    geom_vertices = structure_vertexData(vertices, indices)

    #name = "Geom_{}".format(i)
    create_shape(geom_name, geom_vertices)

    ROBOT_frame.Paste()
    print("{} added to Robot tree".format(geom_name))

--- program Main_Program (robot UR5) ---
  Set Ref.: FrameN
  Set Tool: Gripper
  MoveJ 2 to (0, 0, 0) mm; joints [0, -90, -90, 0, 90, 0]
  MoveJ (csv_data-0)
  Set speed (100.0 mm/s)
  Call Detach
  MoveL (csv_data-1)
  Call Attach
  MoveL (csv_data-2)
  Set speed (300.0 mm/s)
  MoveJ (csv_data-3)
  Set speed (100.0 mm/s)
  MoveL (csv_data-4)
  Call Detach
  MoveL (csv_data-5)
  Set speed (300.0 mm/s)
  MoveJ (csv_data-6)
  Set speed (100.0 mm/s)
  MoveL (csv_data-7)
  Call Attach
  MoveL (csv_data-8)
  Set speed (300.0 mm/s)
  MoveJ (csv_data-9)
  Set speed (100.0 mm/s)
  MoveL (csv_data-10)
  Call Detach
  MoveL (csv_data-11)
  Set speed (300.0 mm/s)
  MoveJ (csv_data-12)
  Set speed (100.0 mm/s)
  MoveL (csv_data-13)
  Call Attach
  MoveL (csv_data-14)
  Set speed (300.0 mm/s)
  MoveJ (csv_data-15)
  Set speed (100.0 mm/s)
  MoveL (csv_data-16)
  Call Detach
  MoveL (csv_data-17)
  Set speed (300.0 mm/s)
  MoveJ (csv_data-18)
  Set speed (100.0 mm/s)
  MoveL (csv_data-19)
  Call Attach
  MoveL (csv_data-20)
  Set speed (300.0 mm/s)
  MoveJ (csv_data-21)
  Set speed (100.0 mm/s)
  MoveL (csv_data-22)
  Call Detach
  MoveL (csv_data-23)
  Set speed (300.0 mm/s)
  MoveJ (csv_data-24)
  Set speed (100.0 mm/s)
  MoveL (csv_data-25)
  Call Attach
  MoveL (csv_data-26)
  Set speed (300.0 mm/s)
  MoveJ (csv_data-27)
  Set speed (100.0 mm/s)
  MoveL (csv_data-28)
  Call Detach
  MoveL (csv_data-29)
  Set speed (300.0 mm/s)
  MoveJ (csv_data-30)
  Set speed (100.0 mm/s)
  MoveL (csv_data-31)
  Call Attach
  MoveL (csv_data-32)
  Set speed (300.0 mm/s)
  MoveJ (csv_data-33)
  Set speed (100.0 mm/s)
  MoveL (csv_data-34)
  Call Detach
  MoveL (csv_data-35)
  Set speed (300.0 mm/s)
  MoveJ (csv_data-36)
  Set speed (100.0 mm/s)
  MoveL (csv_data-37)
  Call Attach
  MoveL (csv_data-38)
  Set speed (300.0 mm/s)
  MoveJ (csv_data-39)
  Set speed (100.0 mm/s)
  MoveL (csv_data-40)
  Call Detach
  MoveL (csv_data-41)
  Set speed (300.0 mm/s)
  MoveJ (csv_data-42)
  Set speed (100.0 mm/s)
  MoveL (csv_data-43)
  Call Attach
  MoveL (csv_data-44)
  Set speed (300.0 mm/s)
  MoveJ (csv_data-45)
  Set speed (100.0 mm/s)
  MoveL (csv_data-46)
  Call Detach
  MoveL (csv_data-47)
  Set speed (300.0 mm/s)
  MoveJ (csv_data-48)
  Set speed (100.0 mm/s)
  MoveL (csv_data-49)
  Call Attach
  MoveL (csv_data-50)
  Set speed (300.0 mm/s)
  MoveJ (csv_data-51)
  Set speed (100.0 mm/s)
  MoveL (csv_data-52)
  Call Detach
  MoveL (csv_data-53)
  Set speed (300.0 mm/s)
  MoveJ (csv_data-54)
  Set speed (100.0 mm/s)
  MoveL (csv_data-55)
  Call Attach
  MoveL (csv_data-56)
  Set speed (300.0 mm/s)
  MoveJ (csv_data-57)
  Set speed (100.0 mm/s)
  MoveL (csv_data-58)
  Call Detach
  MoveL (csv_data-59)
  Set speed (300.0 mm/s)
  MoveJ (csv_data-60)
  Set speed (100.0 mm/s)
  MoveL (csv_data-61)
  Call Attach
  MoveL (csv_data-62)
  Set speed (300.0 mm/s)
  MoveJ (csv_data-63)
  Set speed (100.0 mm/s)
  MoveL (csv_data-64)
  Call Detach
  MoveL (csv_data-65)
  Set speed (300.0 mm/s)
  MoveJ (csv_data-66)
  Set speed (100.0 mm/s)
  MoveL (csv_data-67)
  Call Attach
  MoveL (csv_data-68)
  Set speed (300.0 mm/s)
  MoveJ (csv_data-69)
  Set speed (100.0 mm/s)
  MoveL (csv_data-70)
  Call Detach
  MoveL (csv_data-71)
  Set speed (300.0 mm/s)
  MoveJ (csv_data-72)
  Set speed (100.0 mm/s)
  MoveL (csv_data-73)
  Call Attach
  MoveL (csv_data-74)
  Set speed (300.0 mm/s)
  MoveJ (csv_data-75)
  Set speed (100.0 mm/s)
  MoveL (csv_data-76)
  Call Detach
  MoveL (csv_data-77)
  Set speed (300.0 mm/s)
  MoveJ (csv_data-78)
  Set speed (100.0 mm/s)
  MoveL (csv_data-79)
  Call Attach
  MoveL (csv_data-80)
  Set speed (300.0 mm/s)
  MoveJ (csv_data-81)
  Set speed (100.0 mm/s)
  MoveL (csv_data-82)
  Call Detach
  MoveL (csv_data-83)
  Set speed (300.0 mm/s)
  MoveJ (csv_data-84)
  Set speed (100.0 mm/s)
  MoveL (csv_data-85)
  Call Attach
  MoveL (csv_data-86)
  Set speed (300.0 mm/s)
  MoveJ (csv_data-87)
  Set speed (100.0 mm/s)
  MoveL (csv_data-88)
  Call Detach
  MoveL (csv_data-89)
  Set speed (300.0 mm/s)
  MoveJ (csv_data-90)
  Set speed (100.0 mm/s)
  MoveL (csv_data-91)
  Call Attach
  MoveL (csv_data-92)
  Set speed (300.0 mm/s)
  MoveJ (csv_data-93)
  Set speed (100.0 mm/s)
  MoveL (csv_data-94)
  Call Detach
  MoveL (csv_data-95)
  Set speed (300.0 mm/s)
  MoveJ (csv_data-96)
  Set speed (100.0 mm/s)
  MoveL (csv_data-97)
  Call Attach
  MoveL (csv_data-98)
  Set speed (300.0 mm/s)
  MoveJ (csv_data-99)
  Set speed (100.0 mm/s)
  MoveL (csv_data-100)
  Call Detach
  MoveL (csv_data-101)
  Set speed (300.0 mm/s)
  MoveJ (csv_data-102)
  Set speed (100.0 mm/s)
  MoveL (csv_data-103)
  Call Attach
  MoveL (csv_data-104)
  Set speed (300.0 mm/s)
  MoveJ (csv_data-105)
  Set speed (100.0 mm/s)
  MoveL (csv_data-106)
  Call Detach
  MoveL (csv_data-107)
  Set speed (300.0 mm/s)
  MoveJ (csv_data-108)
  Set speed (100.0 mm/s)
  MoveL (csv_data-109)
  Call Attach
  MoveL (csv_data-110)
  Set speed (300.0 mm/s)
  MoveJ (csv_data-111)
  Set speed (100.0 mm/s)
  MoveL (csv_data-112)
  Call Detach
  MoveL (csv_data-113)
  Set speed (300.0 mm/s)
  MoveJ (csv_data-114)
  Set speed (100.0 mm/s)
  MoveL (csv_data-115)
  Call Attach
  MoveL (csv_data-116)
  Set speed (300.0 mm/s)
  MoveJ (csv_data-117)
  Set speed (100.0 mm/s)
  MoveL (csv_data-118)
  Call Detach
  MoveL (csv_data-119)
  Set speed (300.0 mm/s)
  MoveJ (csv_data-120)
  Set speed (100.0 mm/s)
  MoveL (csv_data-121)
  Call Attach
  MoveL (csv_data-122)
  Set speed (300.0 mm/s)
  MoveJ (csv_data-123)
  Set speed (100.0 mm/s)
  MoveL (csv_data-124)
  Call Detach
  MoveL (csv_data-125)
  Set speed (300.0 mm/s)
  MoveJ (csv_data-126)
  Set speed (100.0 mm/s)
  MoveL (csv_data-127)
  Call Attach
  MoveL (csv_data-128)
  Set speed (300.0 mm/s)
  MoveJ (csv_data-129)
  Set speed (100.0 mm/s)
  MoveL (csv_data-130)
  Call Detach
  MoveL (csv_data-131)
  Set speed (300.0 mm/s)
  MoveJ (csv_data-132)
  Set speed (100.0 mm/s)
  MoveL (csv_data-133)
  Call Attach
  MoveL (csv_data-134)
  Set speed (300.0 mm/s)
  MoveJ (csv_data-135)
  Set speed (100.0 mm/s)
  MoveL (csv_data-136)
  Call Detach
  MoveL (csv_data-137)
  Set speed (300.0 mm/s)
  MoveJ (csv_data-138)
  Set speed (100.0 mm/s)
  MoveL (csv_data-139)
  Call Attach
  MoveL (csv_data-140)
  Set speed (300.0 mm/s)
  MoveJ (csv_data-141)
  Set speed (100.0 mm/s)
  MoveL (csv_data-142)
  Call Detach
  MoveL (csv_data-143)
  Set speed (300.0 mm/s)
  MoveJ (csv_data-144)
  Set speed (100.0 mm/s)
  MoveL (csv_data-145)
  Call Attach
  MoveL (csv_data-146)
  Set speed (300.0 mm/s)
  MoveJ (csv_data-147)
  Set speed (100.0 mm/s)
  MoveL (csv_data-148)
  Call Detach
  MoveL (csv_data-149)
  Set speed (300.0 mm/s)
  MoveJ (csv_data-150)
  Set speed (100.0 mm/s)
  MoveL (csv_data-151)
  Call Attach
  MoveL (csv_data-152)
  Set speed (300.0 mm/s)
  MoveJ (csv_data-153)
  Set speed (100.0 mm/s)
  MoveL (csv_data-154)
  Call Detach
  MoveL (csv_data-155)
  Set speed (300.0 mm/s)
  MoveJ (csv_data-156)
  Set speed (100.0 mm/s)
  MoveL (csv_data-157)
  Call Attach
  MoveL (csv_data-158)
  Set speed (300.0 mm/s)
  MoveJ (csv_data-159)
  Set speed (100.0 mm/s)
  MoveL (csv_data-160)
  Call Detach
  MoveL (csv_data-161)
  Set speed (300.0 mm/s)
  MoveJ (csv_data-162)
  Set speed (100.0 mm/s)
  MoveL (csv_data-163)
  Call Attach
  MoveL (csv_data-164)
  Set speed (300.0 mm/s)
  MoveJ (csv_data-165)
  Set speed (100.0 mm/s)
  MoveL (csv_data-166)
  Call Detach
  MoveL (csv_data-167)
  Set speed (300.0 mm/s)
  MoveJ (csv_data-168)
  Set speed (100.0 mm/s)
  MoveL (csv_data-169)
  Call Attach
  MoveL (csv_data-170)
  Set speed (300.0 mm/s)
  MoveJ (csv_data-171)
  Set speed (100.0 mm/s)
  MoveL (csv_data-172)
  Call Detach
  MoveL (csv_data-173)
  Set speed (300.0 mm/s)
  MoveJ (csv_data-174)
  Set speed (100.0 mm/s)
  MoveL (csv_data-175)
  Call Attach
  MoveL (csv_data-176)
  Set speed (300.0 mm/s)
  MoveJ (csv_data-177)
  Set speed (100.0 mm/s)
  MoveL (csv_data-178)
  Call Detach
  MoveL (csv_data-179)
  Set speed (300.0 mm/s)
  MoveJ 364 to (0, 0, 0) mm; joints [0, -90, -90, 0, 90, 0]

--- program Attach (robot UR5) ---
  Pause 500 ms
  Attach to Gripper
  Pause 500 ms

--- program Detach (robot UR5) ---
  Pause 500 ms
  Detach from Gripper
  Pause 500 ms

--- program Return_Bricks (robot UR5) ---
  Replace objects
